FUNCTION_BLOCK SocketConnectTask IMPLEMENTS ITask
VAR_INPUT
END_VAR
VAR_OUTPUT
END_VAR
VAR
	_execute : BOOL;
	iState: INT;
	_done: BOOL;
	_busy: BOOL;
	_error: BOOL;
	fbSocketConnect : Tc2_TcpIp.FB_SocketConnect;
END_VAR

CASE iState OF
	0:
		IF _execute THEN
			_done := FALSE;
			_busy := TRUE;
			_error := FALSE;
			fbSocketConnect.bExecute := TRUE;
			IF fbSocketConnect.bBusy THEN
				iState := 10;
				_execute := false;
			END_IF
		END_IF
	10:
		IF NOT fbSocketConnect.bBusy THEN
			IF NOT fbSocketConnect.bError THEN
				_done := TRUE;
			ELSE
				_error := TRUE;
			END_IF
			_busy := FALSE;
			fbSocketConnect.bExecute := FALSE;
			iState := 0;
		END_IF
END_CASE

fbSocketConnect(tTimeout := Tc2_System.DEFAULT_ADS_TIMEOUT)

METHOD Abort : BOOL
fbSocketConnect.bExecute := FALSE;
_busy := FALSE;
_execute := FALSE;
Abort := TRUE;
iState := 0;
END_METHOD

PROPERTY Busy : BOOL
GET
Busy := _busy;
END_GET
END_PROPERTY

PROPERTY Done : BOOL
GET
Done := _done;
END_GET
END_PROPERTY

PROPERTY Error : BOOL
GET
Error := _error;
END_GET
END_PROPERTY

METHOD Execute : BOOL
VAR_INPUT
	RemoteIPAddress : Tc2_System.T_IPv4Addr;
	RemotePortNumber : UDINT;
END_VAR
IF NOT fbSocketConnect.bBusy THEN
	fbSocketConnect.sRemoteHost := RemoteIPAddress;
	fbSocketConnect.nRemotePort := RemotePortNumber;	
	Execute := _execute := TRUE;
END_IF
END_METHOD

PROPERTY PUBLIC RemoteSocket : T_HSOCKET
GET
RemoteSocket := fbSocketConnect.hSocket;
END_GET
END_PROPERTY

END_FUNCTION_BLOCK

(* stored: Version 1.1.0.1, ProductVersion 3.1.4024.12
   POU SocketConnectTask: Id {ab0006a8-b1bb-4358-a532-fa52af7574ea}, SpecialFunc None
   Method Abort: Id {b89364ed-0e21-4695-98b8-99b272c7d5b2}
   Property Busy: Id {9c61b440-f4b8-451f-acf6-41b39c2ee667}
   Get Get: Id {abe1cfa3-1c26-4855-8062-aee9127759c1}
   Property Done: Id {c06e83d7-12df-463f-9ef5-32ef1c8f9575}
   Get Get: Id {fa927115-678b-4ec2-8cd6-829673d39909}
   Property Error: Id {7e829a65-c78e-43ac-9b91-7470cfd66cbd}
   Get Get: Id {1f526684-2b40-4ae2-94ea-b3647a444046}
   Method Execute: Id {99fabac9-6396-449b-a6fb-a610ff7ef49b}
   Property RemoteSocket: Id {fa38ac05-03cc-4c98-aef0-de370d43d756}
   Get Get: Id {f45f28ac-1b65-43bf-93ad-53fb7683bede} *)
